FUNCTION_BLOCK Test_AggregateResult_Error EXTENDS T_UnitTestBase
VAR
	ResultAggregate : T_ResultAggregate;
	Execution1 : T_Execution;
	Execution2 : T_Execution;
	Execution3 : T_Execution;
END_VAR

METHOD Init
SUPER^.Init();

Execution1.FB_init(FALSE,FALSE);
Execution2.FB_init(FALSE,FALSE);
Execution3.FB_init(FALSE,FALSE);
END_METHOD

{attribute 'analysis' := '-33'} // inhibit unused variable warning
METHOD RunTest
ResultAggregate.ClearResults();

ResultAggregate.AddResult(Execution1);
ResultAggregate.AddResult(Execution2);
ResultAggregate.AddResult(Execution3);

Execution1.Start();
Execution1.SetBusy();

AssertIsTrue(Condition := ResultAggregate.Error = FALSE,
             Message   := 'ResultAggregate.Error is not false');

Execution3.Start();
Execution3.SetBusy();
Execution3.SetError('Error Message');

AssertIsTrue(Condition := ResultAggregate.Error = TRUE,
             Message   := 'ResultAggregate.Error is false');

TestCompleted := TRUE;
END_METHOD

END_FUNCTION_BLOCK

(* stored: Version 1.1.0.1, ProductVersion 3.1.4024.12
   POU Test_AggregateResult_Error: Id {2cc1540d-06bd-4742-a6db-1ca1c7513675}, SpecialFunc None
   Method Init: Id {2ebfb763-8f5f-4d4a-b7e6-afe836ec19bc}
   Method RunTest: Id {8df4aa35-d688-4c72-8ddd-5f355b6b1baa} *)
